(* PLC project Senza_nome, Sconosciuto Senza_nome 1 *)
(* stored: creationDateTime 2020-08-24T19:28:07, modificationDateTime 2020-09-29T15:52:42 *)

FUNCTION_BLOCK TP_WITH_RESET
  VAR_INPUT
    IN : BOOL;
    PT : TIME;
    RESET : BOOL;
  END_VAR
  VAR_OUTPUT
    Q : BOOL;
    ET : TIME := T#0s;
  END_VAR
  VAR
    STATE : SINT := 0;
    PREV_IN : BOOL := FALSE;
    CURRENT_TIME : TIME;
    START_TIME : TIME;
  END_VAR

            (* Pragma to set current time *)
{__SET_VAR(data__->,CURRENT_TIME,,__CURRENT_TIME)}

(*Timer block code *)
IF ((STATE = 0) AND NOT(PREV_IN) AND IN) THEN  (* found rising edge on IN *)
    (* start timer... *)
    STATE := 1;
    Q := TRUE;
    START_TIME := CURRENT_TIME;

ELSIF (STATE = 1) THEN (* timer counting *)
    IF ((START_TIME + PT) <= CURRENT_TIME) THEN (* timer expired *)
        STATE := 2;
        Q := FALSE;
        ET := PT;
    ELSE (* continue counting *)
        ET := CURRENT_TIME - START_TIME;
    END_IF;
END_IF;

IF ((STATE = 2) AND NOT(IN)) THEN
    ET := T#0s;
    STATE := 0;
END_IF;

IF (RESET) THEN (* reset pressed *)
  ET := T#0s;
  STATE := 0;
  Q := FALSE;
END_IF;

PREV_IN := IN;
          
END_FUNCTION_BLOCK

FUNCTION_BLOCK AccensioneProgrammata
  VAR
    TP_WITH_RESET0 : TP_WITH_RESET;  (* Istanza blocco funzionale timer con reset *)
    Aux : BOOL;  (* Variabile ausiliare *)
    Tempo0 : TIME := T#3s;  (* Variabile connessa all'accensione programmata *)
  END_VAR
  VAR_INPUT
    OreDallAccensione : TIME;  (* Associata al PT del secondo timer *)
    Ingresso : BOOL;  (* Variabile di ingresso *)
    Reset : BOOL;  (* Variabile connessa al reset dei timer *)
  END_VAR
  VAR_OUTPUT
    UscitaOn : BOOL;  (* Variabile di uscita *)
  END_VAR
  VAR
    TP_WITH_RESET1 : TP_WITH_RESET;  (* Istanza blocco funzionale timer con reset *)
  END_VAR
  VAR  (* added by the conversion: wires and edge detectors of the diagram *)
    R_TRIG1 : R_TRIG;
    R_TRIG2 : R_TRIG;
    F_TRIG3 : F_TRIG;
  END_VAR

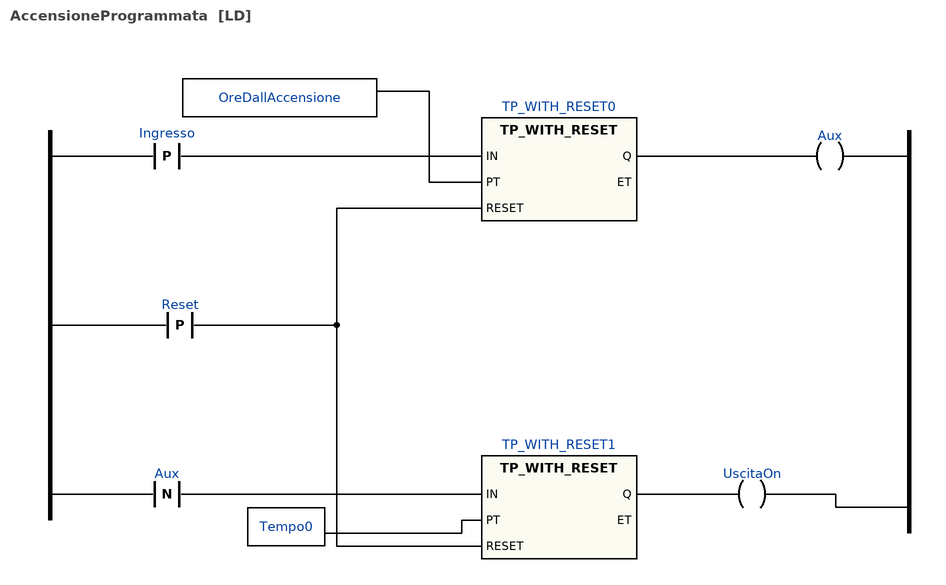
(* LD diagram, written out as Structured Text *)
R_TRIG1(CLK := Ingresso);
R_TRIG2(CLK := Reset);
TP_WITH_RESET0(IN := R_TRIG1.Q, PT := OreDallAccensione, RESET := R_TRIG2.Q);
Aux := TP_WITH_RESET0.Q;
F_TRIG3(CLK := Aux);
TP_WITH_RESET1(IN := F_TRIG3.Q, PT := Tempo0, RESET := R_TRIG2.Q);
UscitaOn := TP_WITH_RESET1.Q;
END_FUNCTION_BLOCK

FUNCTION_BLOCK Macchine
  VAR_INPUT
    TempoDiLavorazione : TIME;  (* Variabile connessa al tempo di lavorazione della macchina *)
    Ingresso : BOOL := 0;  (* Variabile di ingresso *)
    Reset : BOOL := 0;  (* Variabile connessa al reset dei timer *)
  END_VAR
  VAR_OUTPUT
    UscitaMacchina : BOOL := 0;  (* Variabile di uscita *)
  END_VAR
  VAR
    TP_WITH_RESET0 : TP_WITH_RESET;  (* Istanza blocco funzionale timer con reset *)
  END_VAR
  VAR  (* added by the conversion: wires and edge detectors of the diagram *)
    R_TRIG1 : R_TRIG;
    R_TRIG2 : R_TRIG;
  END_VAR

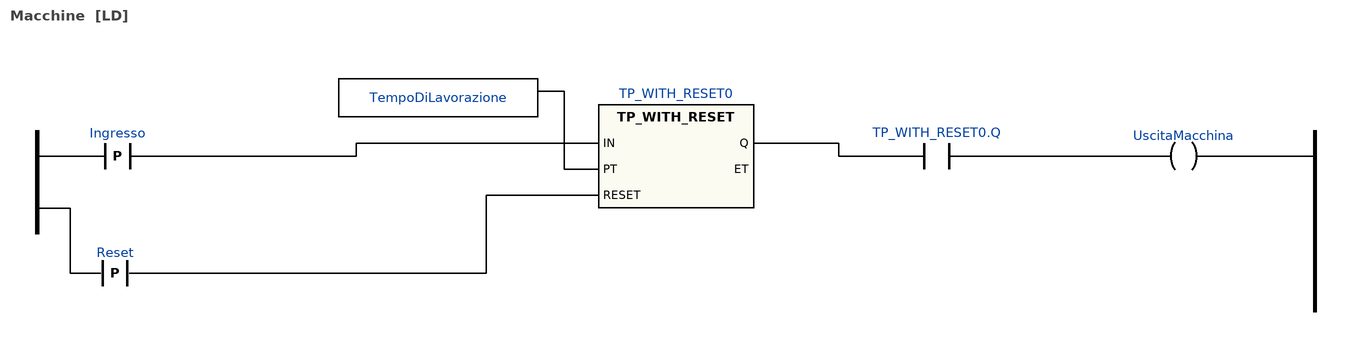
(* LD diagram, written out as Structured Text *)
R_TRIG1(CLK := Ingresso);
R_TRIG2(CLK := Reset);
TP_WITH_RESET0(IN := R_TRIG1.Q, PT := TempoDiLavorazione, RESET := R_TRIG2.Q);
UscitaMacchina := TP_WITH_RESET0.Q AND TP_WITH_RESET0.Q;
END_FUNCTION_BLOCK

FUNCTION_BLOCK Nastro1
  VAR_INPUT
    TempoEsecuzione : TIME;  (* Variabile connessa al tempo di movimento del nastro *)
  END_VAR
  VAR
    TempoInterno : TIME := T#2s;  (* Associata al PT del primo timer *)
  END_VAR
  VAR_INPUT
    Ingresso : BOOL := 0;  (* Variabile di ingresso *)
    reset : BOOL := 0;  (* Variabile connessa al reset dei timer *)
  END_VAR
  VAR_OUTPUT
    UscitaNastro : BOOL := 0;  (* Variabile di uscita *)
  END_VAR
  VAR
    aux : BOOL;  (* Variabile ausiliare *)
    TP_WITH_RESET1 : TP_WITH_RESET;  (* Istanza blocco funzionale timer con reset *)
    TP_WITH_RESET2 : TP_WITH_RESET;  (* Istanza blocco funzionale timer con reset *)
  END_VAR
  VAR  (* added by the conversion: wires and edge detectors of the diagram *)
    R_TRIG1 : R_TRIG;
    R_TRIG2 : R_TRIG;
    F_TRIG3 : F_TRIG;
  END_VAR

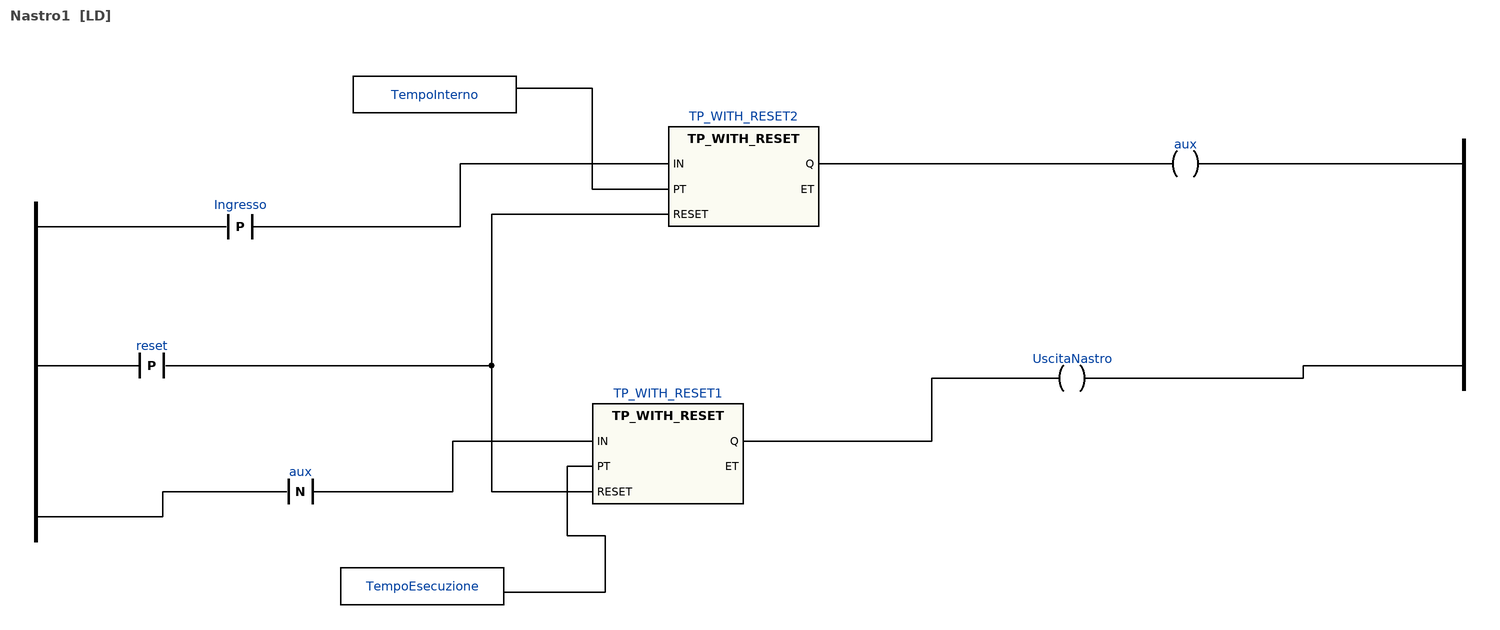
(* LD diagram, written out as Structured Text *)
R_TRIG1(CLK := Ingresso);
R_TRIG2(CLK := reset);
TP_WITH_RESET2(IN := R_TRIG1.Q, PT := TempoInterno, RESET := R_TRIG2.Q);
aux := TP_WITH_RESET2.Q;
F_TRIG3(CLK := aux);
TP_WITH_RESET1(IN := F_TRIG3.Q, PT := TempoEsecuzione, RESET := R_TRIG2.Q);
UscitaNastro := TP_WITH_RESET1.Q;
END_FUNCTION_BLOCK

FUNCTION_BLOCK RisprmioEnergetico
  VAR_OUTPUT
    Uscita : BOOL := 0;  (* Variabile di uscita *)
  END_VAR
  VAR
    aux : BOOL := 0;  (* Variabile ausiliare *)
  END_VAR
  VAR_INPUT
    Ingresso : BOOL := 0;  (* Variabile di ingresso *)
    Reset : BOOL := 0;  (* Variabile connessa al reset dei timer *)
    Tempo : TIME;  (* Associata al PT del primo timer *)
  END_VAR
  VAR
    Tempo2 : TIME := T#4s;  (* Associata al PT del secondo timer *)
    TP_WITH_RESET0 : TP_WITH_RESET;  (* Istanza blocco funzionale timer con reset *)
    TP_WITH_RESET1 : TP_WITH_RESET;  (* Istanza blocco funzionale timer con reset *)
  END_VAR
  VAR  (* added by the conversion: wires and edge detectors of the diagram *)
    R_TRIG1 : R_TRIG;
    F_TRIG2 : F_TRIG;
  END_VAR

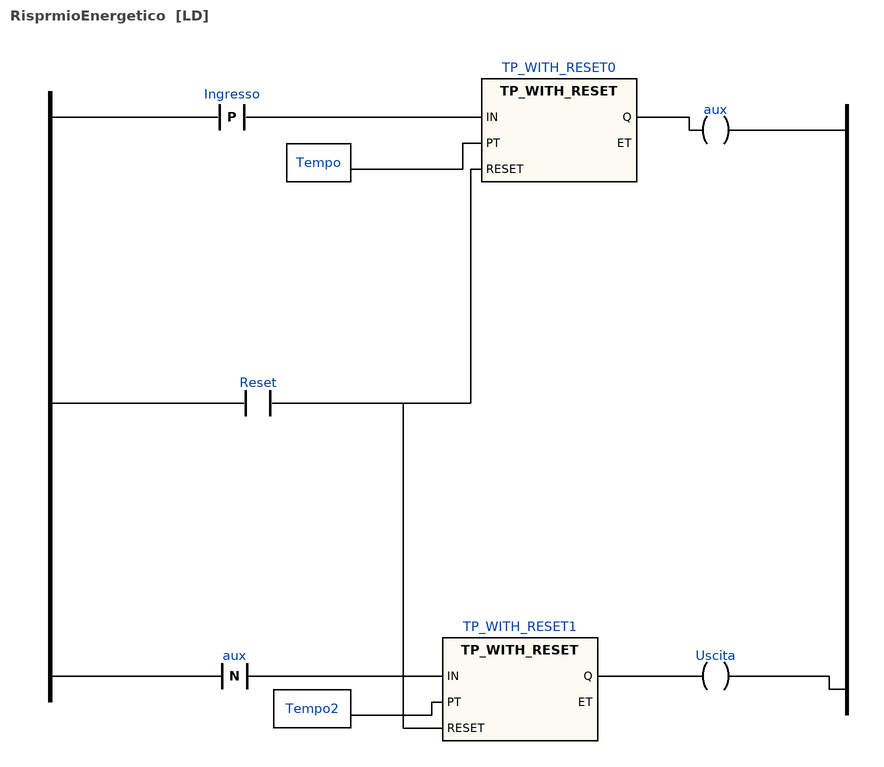
(* LD diagram, written out as Structured Text *)
R_TRIG1(CLK := Ingresso);
TP_WITH_RESET0(IN := R_TRIG1.Q, PT := Tempo, RESET := Reset);
aux := TP_WITH_RESET0.Q;
F_TRIG2(CLK := aux);
TP_WITH_RESET1(IN := F_TRIG2.Q, PT := Tempo2, RESET := Reset);
Uscita := TP_WITH_RESET1.Q;
END_FUNCTION_BLOCK

PROGRAM program0
  VAR
    TastoOn : BOOL := 0;  (* Variabile connessa al pulsante On della macchina *)
  END_VAR
  VAR RETAIN
    AccensioneMan : BOOL := 0;  (* Variabile connessa all'accensione con modalità manuale della macchina *)
    AccensioneAut : BOOL := 0;  (* Variabile connessa all'accensione con modalità automatica della macchina *)
  END_VAR
  VAR
    RipristinoX : BOOL := 0;  (* Replica (per problemi di open plc) il marker di fase della fase Ripristino *)
    RisparmioEnergetico1 : BOOL := 0;  (* Variabile per risparimio energetico 1 *)
    RisparmioEnergetico2 : BOOL := 0;  (* Variabile per risparimio energetico 2 *)
    AttivaReset : BOOL := 0;  (* Attiva il reset del timer *)
    AttivaResetRipr : BOOL := 0;  (* Attiva il reset del timer *)
    AttivaReset0 : BOOL := 0;  (* Attiva il reset del timer *)
    AttivaReset2 : BOOL := 0;  (* Attiva il reset del timer *)
    AttivaReset3 : BOOL := 0;  (* Attiva il reset del timer *)
    AttivaReset4 : BOOL := 0;  (* Attiva il reset del timer *)
    AttivaReset5 : BOOL := 0;  (* Attiva il reset del timer *)
    AttivaReset6 : BOOL := 0;  (* Attiva il reset del timer *)
    AttivaReset7 : BOOL := 0;  (* Attiva il reset del timer *)
    TempoAttesa : BOOL := 0;  (* Sono utilizzate in sostituzione ai timer di fase *)
    TempoAttesa2 : BOOL := 0;  (* Sono utilizzate in sostituzione ai timer di fase *)
    TempoAttesa3 : BOOL := 0;  (* Sono utilizzate in sostituzione ai timer di fase *)
    TimeDummy1 : BOOL := 0;  (* Sono utilizzate in sostituzione ai timer di fase *)
    TimeDummy2 : BOOL := 0;  (* Sono utilizzate in sostituzione ai timer di fase *)
    TimeDummy3 : BOOL := 0;  (* Sono utilizzate in sostituzione ai timer di fase *)
    TimeDummy4 : BOOL := 0;  (* Sono utilizzate in sostituzione ai timer di fase *)
    TimeDummy5 : BOOL := 0;  (* Sono utilizzate in sostituzione ai timer di fase *)
    TimeDummy6 : BOOL := 0;  (* Sono utilizzate in sostituzione ai timer di fase *)
    TimeDummy7 : BOOL := 0;  (* Sono utilizzate in sostituzione ai timer di fase *)
    MacchinaRiscaldata : BOOL := 0;  (* Variabile associata al riscaldamento iniziale della macchina *)
    Time3 : TIME := T#5s;  (* Varibile di tempo utilizzata in Nastro1 e preFineNastro *)
    Time5 : TIME := T#7s;  (* Varibile di tempo utilizzata in fust,Nastro2,StampaAcaldo *)
    Time6 : TIME := T#12s;  (* Varibile di tempo utilizzata in SvuotaNastro *)
    Time7 : TIME := T#900s;  (* Varibile di tempo utilizzata in SvuotaNastro *)
    Time8 : TIME := T#1h;  (* Varibile di tempo utilizzata in SvuotaNastro *)
    Time9 : TIME := T#60s;  (* Varibile di tempo utilizzata in SvuotaNastro *)
  END_VAR
  VAR RETAIN
    TempoProgrammato : TIME := T#0s;  (* Tempo inserito per la futura accensione programmata *)
  END_VAR
  VAR
    LedVerde : BOOL := 0;  (* Variabile connessa al led verde *)
    LedGiallo : BOOL := 0;  (* Variabile connessa al led giallo *)
    LedBianco : BOOL := 0;  (* Variabile connessa al led bianco *)
    ErroreMacchina2 : BOOL := 0;  (* Variabile connessa ad un errore alla macchina che stampa a caldo *)
    ErroreMacchina1 : BOOL := 0;  (* Variabile connessa ad un errore alla macchina che fustella *)
    LedNero : BOOL := 0;  (* Variabile connessa al led nero *)
    LedRosso : BOOL := 0;  (* Variabile connessa al led rosso *)
    TastoCaricoBusta : BOOL := 0;  (* Variabile connessa al pulsante Carico Busta *)
    TastoOff : BOOL := 0;  (* Variabile connessa al pulsante Off della macchina *)
    StartLavorazione : BOOL := 0;  (* Variabile connessa al pulsante Start Lavorazione *)
    Vano : BOOL := 1;  (* Variabile legata al vano di sicurezza della macchina ( gestita in logica negata) *)
    TastoEmergenza : BOOL := 1;  (* Variabile connessa al pulsante di Emergenza della macchina ( gestita in logica negata) *)
    StatoFustellatrice : BOOL := 0;  (* Variabile connessa allo stato della Fustellatrice *)
    StatoStampaACaldo : BOOL := 0;  (* Variabile connessa allo stato della stampa a caldo *)
    Nastro : BOOL := 0;  (* Variabile connessa al nastro trasportatore *)
    SensoreFoil : BOOL := 0;  (* Variabile connessa al sensore del foil (inchiostro) della stampa a caldo *)
    SensoreTemp : BOOL := 0;  (* Variabile connessa al sensore della temperatura della stampa a caldo *)
    SensoreLama : BOOL := 0;  (* Variabile connessa al sensore della lama (indica l'usura) della fustellatrice *)
    RisprmioEnergetico1 : RisprmioEnergetico;  (* Istanza blocco funzionale *)
    RisprmioEnergetico0 : RisprmioEnergetico;  (* Istanza blocco funzionale *)
    Nastro11 : Nastro1;  (* Istanza blocco funzionale *)
    Macchine0 : Macchine;  (* Istanza blocco funzionale *)
    Macchine1 : Macchine;  (* Istanza blocco funzionale *)
    Nastro12 : Nastro1;  (* Istanza blocco funzionale *)
    Nastro10 : Nastro1;  (* Istanza blocco funzionale *)
    AccensioneProgrammata0 : AccensioneProgrammata;  (* Istanza blocco funzionale *)
    Nastro13 : Nastro1;  (* Istanza blocco funzionale *)
    TP0 : TP;
    TP1 : TP;
    RisprmioEnergetico2 : RisprmioEnergetico;
    TP2 : TP;
  END_VAR
  VAR  (* added by the conversion: wires and edge detectors of the diagram *)
    F_TRIG1 : F_TRIG;
    F_TRIG2 : F_TRIG;
  END_VAR

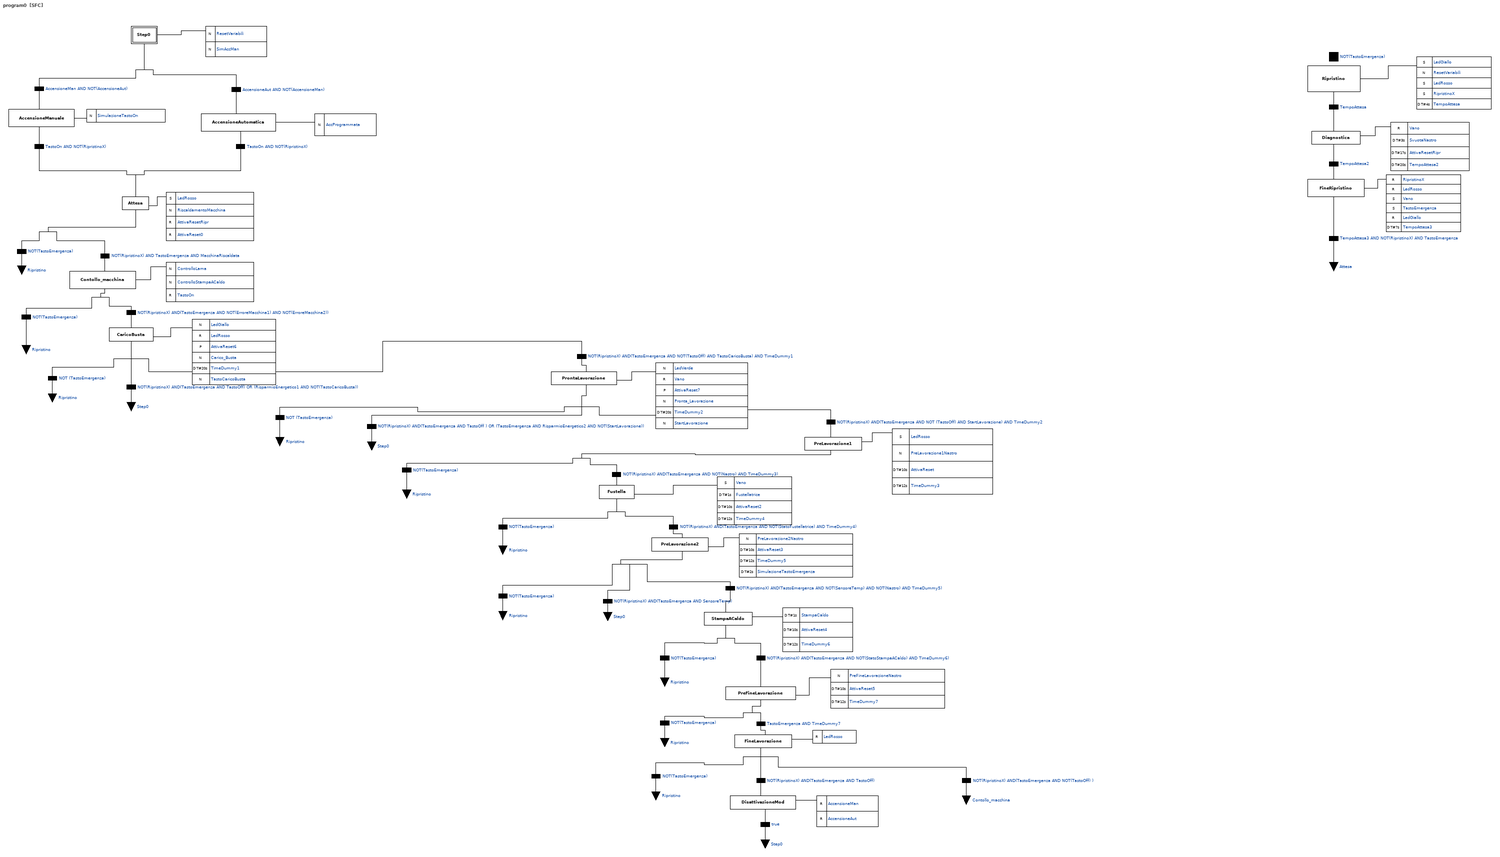
INITIAL_STEP Step0:
  ResetVariabili(N);
  SimAccMan(N);
END_STEP
TRANSITION FROM Step0 TO AccensioneManuale
  := AccensioneMan AND NOT(AccensioneAut);
END_TRANSITION
TRANSITION FROM Step0 TO AccensioneAutomatica
  := AccensioneAut AND NOT(AccensioneMan);
END_TRANSITION
STEP Ripristino:
  LedGiallo(S);
  ResetVariabili(N);
  LedRosso(S);
  RipristinoX(S);
  TempoAttesa(D, T#4s);
END_STEP
TRANSITION FROM Ripristino TO Diagnostica
  := TempoAttesa;
END_TRANSITION
STEP AccensioneManuale:
  SimulazioneTastoOn(N);
END_STEP
TRANSITION FROM AccensioneManuale TO Attesa
  := TastoOn AND NOT(RipristinoX);
END_TRANSITION
STEP AccensioneAutomatica:
  AccProgrammata(N);
END_STEP
TRANSITION FROM AccensioneAutomatica TO Attesa
  := TastoOn AND NOT(RipristinoX);
END_TRANSITION
STEP Diagnostica:
  Vano(R);
  SvuotaNastro(D, T#3s);
  AttivaResetRipr(D, T#17s);
  TempoAttesa2(D, T#20s);
END_STEP
TRANSITION FROM Diagnostica TO FineRipristino
  := TempoAttesa2;
END_TRANSITION
STEP FineRipristino:
  RipristinoX(R);
  LedRosso(R);
  Vano(S);
  TastoEmergenza(S);
  LedGiallo(R);
  TempoAttesa3(D, T#7s);
END_STEP
TRANSITION FROM FineRipristino TO Attesa
  := TempoAttesa3 AND NOT(RipristinoX) AND TastoEmergenza;
END_TRANSITION
STEP Attesa:
  LedRosso(S);
  RiscaldamentoMacchina(N);
  AttivaResetRipr(R);
  AttivaReset0(R);
END_STEP
TRANSITION FROM Attesa TO Ripristino
  := NOT(TastoEmergenza);
END_TRANSITION
TRANSITION FROM Attesa TO Contollo_macchina
  := NOT(RipristinoX) AND TastoEmergenza AND MacchinaRiscaldata;
END_TRANSITION
STEP Contollo_macchina:
  ControlloLama(N);
  ControlloStampaACaldo(N);
  TastoOn(R);
END_STEP
TRANSITION FROM Contollo_macchina TO Ripristino
  := NOT(TastoEmergenza);
END_TRANSITION
TRANSITION FROM Contollo_macchina TO CaricoBusta
  := NOT(RipristinoX) AND(TastoEmergenza AND NOT(ErroreMacchina1) AND NOT(ErroreMacchina2));
END_TRANSITION
STEP CaricoBusta:
  LedGiallo(N);
  LedRosso(R);
  AttivaReset6(P);
  Carico_Busta(N);
  TimeDummy1(D, T#20s);
  TastoCaricoBusta(N);
END_STEP
TRANSITION FROM CaricoBusta TO Ripristino
  := NOT (TastoEmergenza);
END_TRANSITION
TRANSITION FROM CaricoBusta TO Step0
  := NOT(RipristinoX) AND(TastoEmergenza AND TastoOff) OR (RisparmioEnergetico1 AND NOT(TastoCaricoBusta));
END_TRANSITION
TRANSITION FROM CaricoBusta TO ProntaLavorazione
  := NOT(RipristinoX) AND(TastoEmergenza AND NOT(TastoOff) AND TastoCaricoBusta) AND TimeDummy1;
END_TRANSITION
STEP ProntaLavorazione:
  LedVerde(N);
  Vano(R);
  AttivaReset7(P);
  Pronta_Lavorazione(N);
  TimeDummy2(D, T#20s);
  StartLavorazione(N);
END_STEP
TRANSITION FROM ProntaLavorazione TO Ripristino
  := NOT (TastoEmergenza);
END_TRANSITION
TRANSITION FROM ProntaLavorazione TO Step0
  := NOT(RipristinoX) AND(TastoEmergenza AND TastoOff ) OR (TastoEmergenza AND RisparmioEnergetico2 AND NOT(StartLavorazione));
END_TRANSITION
TRANSITION FROM ProntaLavorazione TO PreLavorazione1
  := NOT(RipristinoX) AND(TastoEmergenza AND NOT (TastoOff) AND StartLavorazione) AND TimeDummy2;
END_TRANSITION
STEP PreLavorazione1:
  LedRosso(S);
  PreLavorazione1Nastro(N);
  AttivaReset(D, T#10s);
  TimeDummy3(D, T#12s);
END_STEP
TRANSITION FROM PreLavorazione1 TO Ripristino
  := NOT(TastoEmergenza);
END_TRANSITION
TRANSITION FROM PreLavorazione1 TO Fustella
  := NOT(RipristinoX) AND(TastoEmergenza AND NOT(Nastro) AND TimeDummy3);
END_TRANSITION
STEP Fustella:
  Vano(S);
  Fustellatrice(D, T#1s);
  AttivaReset2(D, T#10s);
  TimeDummy4(D, T#12s);
END_STEP
TRANSITION FROM Fustella TO Ripristino
  := NOT(TastoEmergenza);
END_TRANSITION
TRANSITION FROM Fustella TO PreLavorazione2
  := NOT(RipristinoX) AND(TastoEmergenza AND NOT(StatoFustellatrice) AND TimeDummy4);
END_TRANSITION
STEP PreLavorazione2:
  PreLavorazione2Nastro(N);
  AttivaReset3(D, T#10s);
  TimeDummy5(D, T#12s);
  SimulazioneTastoEmergenza(D, T#2s);
END_STEP
TRANSITION FROM PreLavorazione2 TO Ripristino
  := NOT(TastoEmergenza);
END_TRANSITION
TRANSITION FROM PreLavorazione2 TO StampaACaldo
  := NOT(RipristinoX) AND(TastoEmergenza AND NOT(SensoreTemp) AND NOT(Nastro) AND TimeDummy5);
END_TRANSITION
TRANSITION FROM PreLavorazione2 TO Step0
  := NOT(RipristinoX) AND(TastoEmergenza AND SensoreTemp);
END_TRANSITION
STEP StampaACaldo:
  StampaCaldo(D, T#1s);
  AttivaReset4(D, T#10s);
  TimeDummy6(D, T#12s);
END_STEP
TRANSITION FROM StampaACaldo TO Ripristino
  := NOT(TastoEmergenza);
END_TRANSITION
TRANSITION FROM StampaACaldo TO PreFineLavorazione
  := NOT(RipristinoX) AND(TastoEmergenza AND NOT(StatoStampaACaldo) AND TimeDummy6);
END_TRANSITION
STEP PreFineLavorazione:
  PreFineLavorazioneNastro(N);
  AttivaReset5(D, T#10s);
  TimeDummy7(D, T#12s);
END_STEP
TRANSITION FROM PreFineLavorazione TO FineLavorazione
  := TastoEmergenza AND TimeDummy7;
END_TRANSITION
TRANSITION FROM PreFineLavorazione TO Ripristino
  := NOT(TastoEmergenza);
END_TRANSITION
STEP FineLavorazione:
  LedRosso(R);
END_STEP
TRANSITION FROM FineLavorazione TO Ripristino
  := NOT(TastoEmergenza);
END_TRANSITION
TRANSITION FROM FineLavorazione TO DisattivazioneMod
  := NOT(RipristinoX) AND(TastoEmergenza AND TastoOff);
END_TRANSITION
TRANSITION FROM FineLavorazione TO Contollo_macchina
  := NOT(RipristinoX) AND(TastoEmergenza AND NOT(TastoOff) );
END_TRANSITION
STEP DisattivazioneMod:
  AccensioneMan(R);
  AccensioneAut(R);
END_STEP
TRANSITION FROM DisattivazioneMod TO Step0
  := true;
END_TRANSITION
TRANSITION FROM ? TO ?
  := NOT(TastoEmergenza);
END_TRANSITION

ACTION RiscaldamentoMacchina:
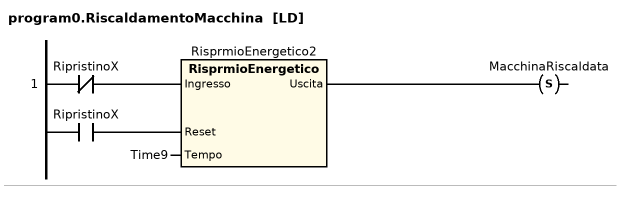
(* LD diagram, written out as Structured Text *)
RisprmioEnergetico2(Ingresso := NOT RipristinoX, Reset := RipristinoX, Tempo := Time9);
IF RisprmioEnergetico2.Uscita THEN MacchinaRiscaldata := TRUE; END_IF;
END_ACTION

ACTION ControlloLama:
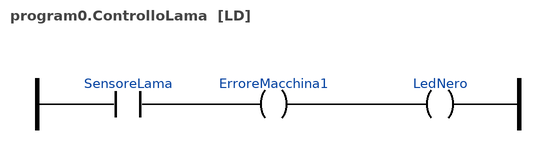
(* LD diagram, written out as Structured Text *)
ErroreMacchina1 := SensoreLama;
LedNero := SensoreLama;
END_ACTION

ACTION ControlloStampaACaldo:
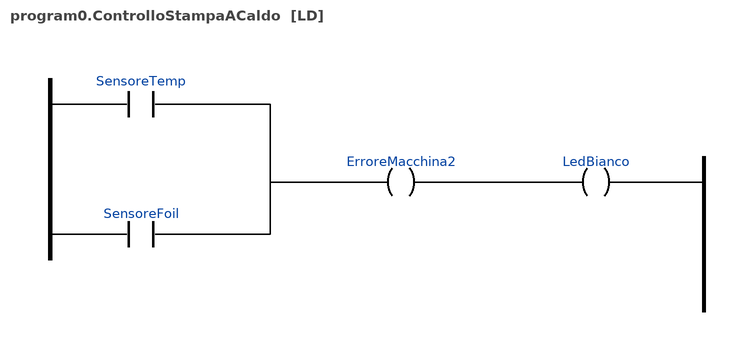
(* LD diagram, written out as Structured Text *)
ErroreMacchina2 := SensoreTemp OR SensoreFoil;
LedBianco := SensoreTemp OR SensoreFoil;
END_ACTION

ACTION Carico_Busta:
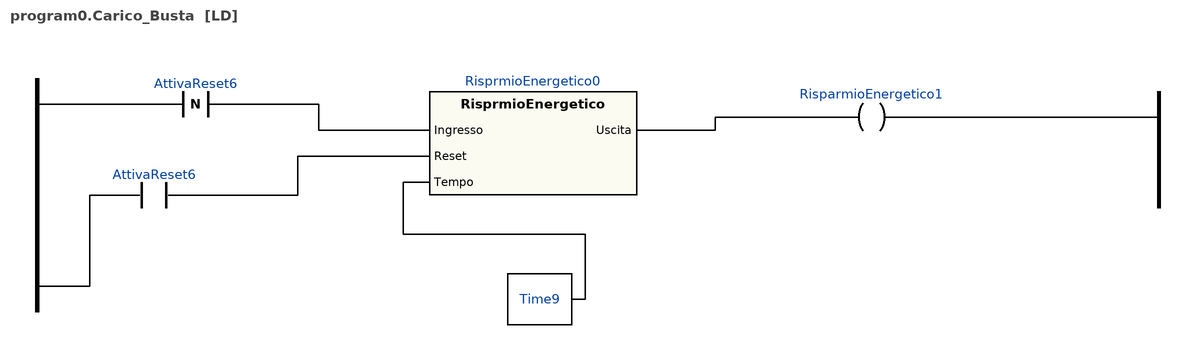
(* LD diagram, written out as Structured Text *)
F_TRIG1(CLK := AttivaReset6);
RisprmioEnergetico0(Ingresso := F_TRIG1.Q, Reset := AttivaReset6, Tempo := Time9);
RisparmioEnergetico1 := RisprmioEnergetico0.Uscita;
END_ACTION

ACTION Pronta_Lavorazione:
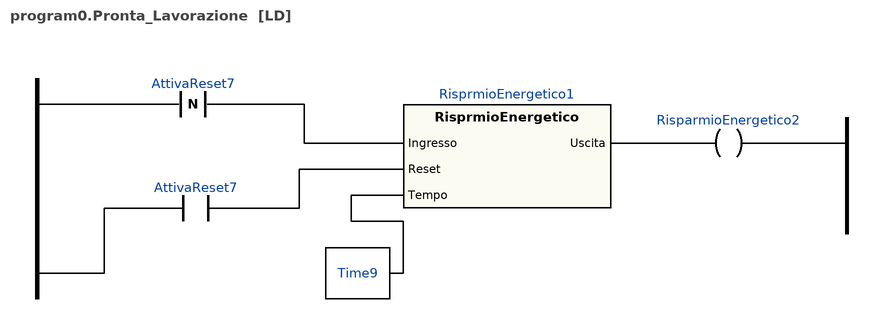
(* LD diagram, written out as Structured Text *)
F_TRIG2(CLK := AttivaReset7);
RisprmioEnergetico1(Ingresso := F_TRIG2.Q, Reset := AttivaReset7, Tempo := Time9);
RisparmioEnergetico2 := RisprmioEnergetico1.Uscita;
END_ACTION

ACTION PreLavorazione1Nastro:
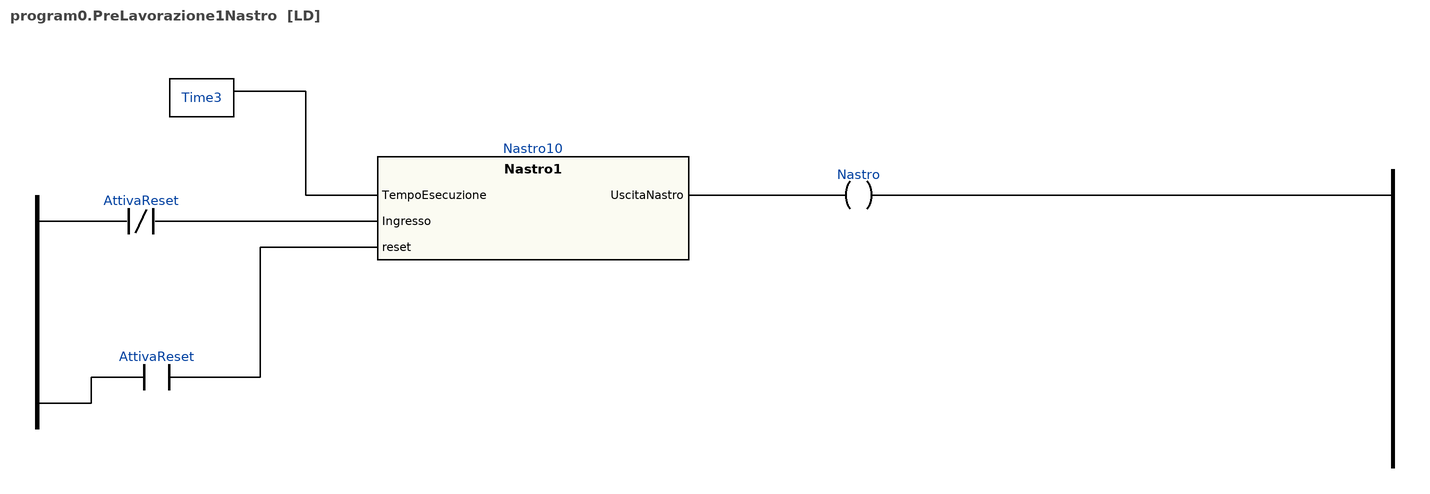
(* LD diagram, written out as Structured Text *)
Nastro10(TempoEsecuzione := Time3, Ingresso := NOT AttivaReset, reset := AttivaReset);
Nastro := Nastro10.UscitaNastro;
END_ACTION

ACTION Fustellatrice:
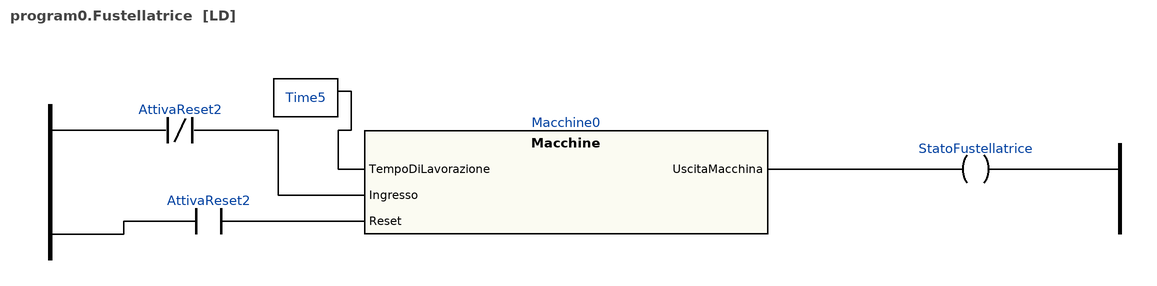
(* LD diagram, written out as Structured Text *)
Macchine0(TempoDiLavorazione := Time5, Ingresso := NOT AttivaReset2, Reset := AttivaReset2);
StatoFustellatrice := Macchine0.UscitaMacchina;
END_ACTION

ACTION PreLavorazione2Nastro:
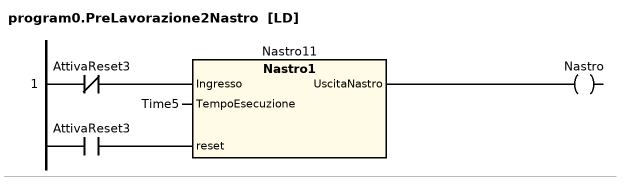
(* LD diagram, written out as Structured Text *)
Nastro11(TempoEsecuzione := Time5, Ingresso := NOT AttivaReset3, reset := AttivaReset3);
Nastro := Nastro11.UscitaNastro;
END_ACTION

ACTION StampaCaldo:
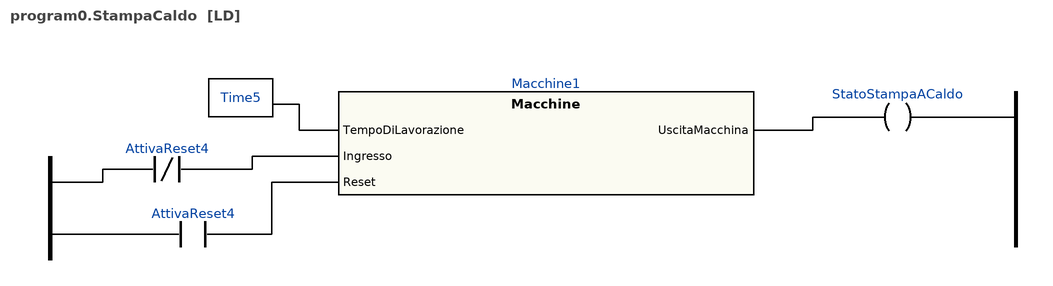
(* LD diagram, written out as Structured Text *)
Macchine1(TempoDiLavorazione := Time5, Ingresso := NOT AttivaReset4, Reset := AttivaReset4);
StatoStampaACaldo := Macchine1.UscitaMacchina;
END_ACTION

ACTION ResetVariabili:
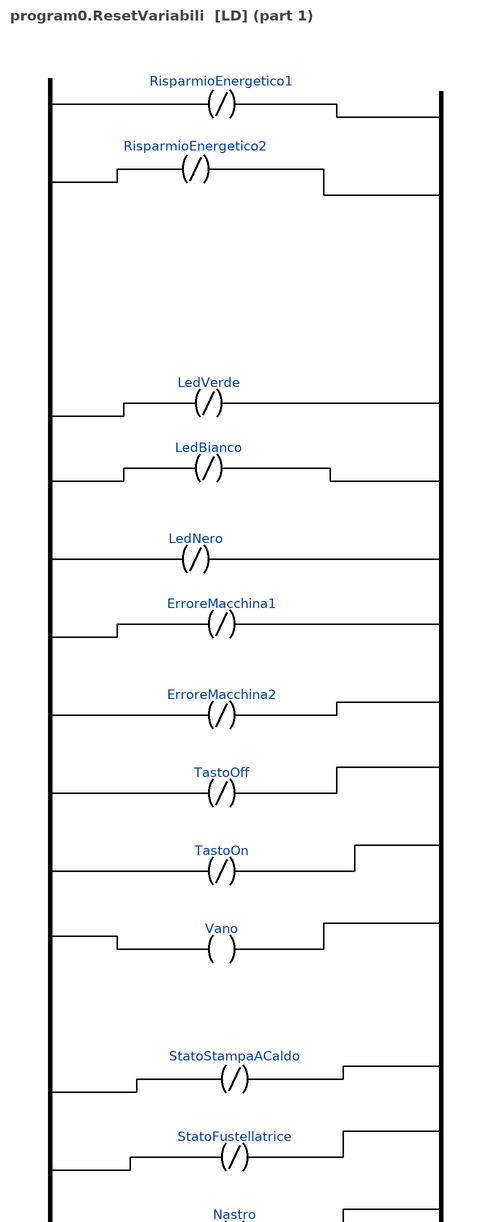
(* LD diagram, written out as Structured Text *)
RisparmioEnergetico1 := NOT TRUE;
RisparmioEnergetico2 := NOT TRUE;
LedVerde := NOT TRUE;
LedBianco := NOT TRUE;
LedNero := NOT TRUE;
ErroreMacchina1 := NOT TRUE;
ErroreMacchina2 := NOT TRUE;
TastoOff := NOT TRUE;
TastoOn := NOT TRUE;
Vano := TRUE;
StatoStampaACaldo := NOT TRUE;
StatoFustellatrice := NOT TRUE;
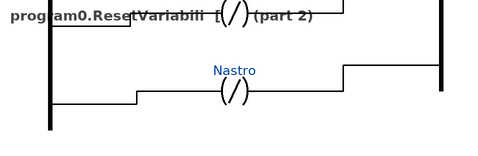
Nastro := NOT TRUE;
END_ACTION

ACTION SpegniRipristino:
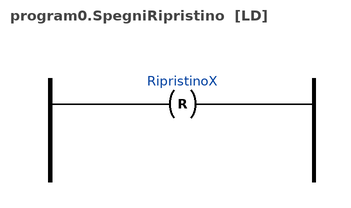
(* LD diagram, written out as Structured Text *)
IF TRUE THEN RipristinoX := FALSE; END_IF;
END_ACTION

ACTION SpegniTasti:
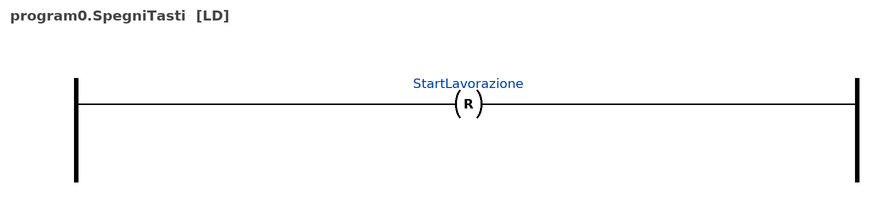
(* LD diagram, written out as Structured Text *)
IF TRUE THEN StartLavorazione := FALSE; END_IF;
END_ACTION

ACTION PreFineLavorazioneNastro:
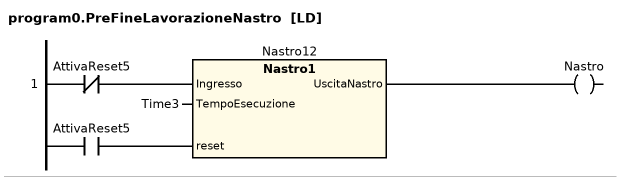
(* LD diagram, written out as Structured Text *)
Nastro12(TempoEsecuzione := Time3, Ingresso := NOT AttivaReset5, reset := AttivaReset5);
Nastro := Nastro12.UscitaNastro;
END_ACTION

ACTION AccProgrammata:
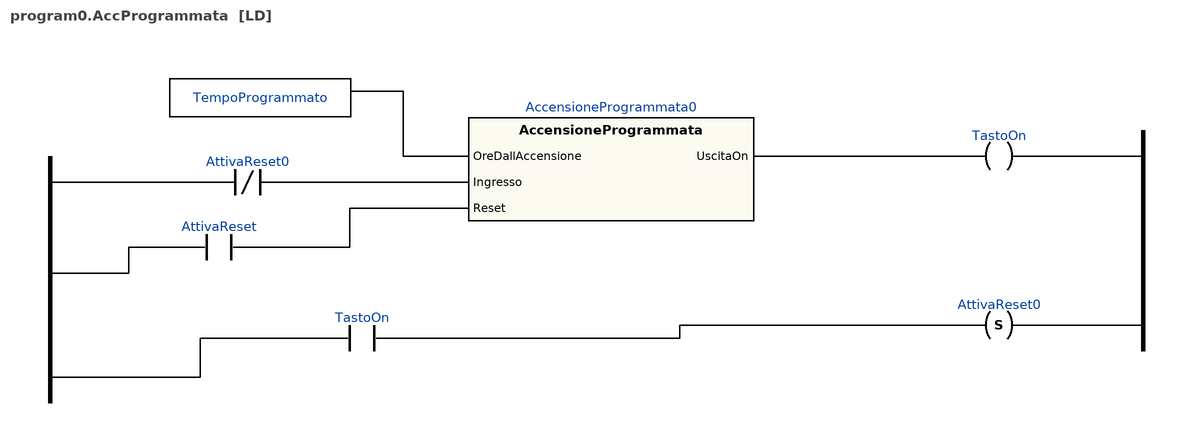
(* LD diagram, written out as Structured Text *)
AccensioneProgrammata0(OreDallAccensione := TempoProgrammato, Ingresso := NOT AttivaReset0, Reset := AttivaReset);
TastoOn := AccensioneProgrammata0.UscitaOn;
IF TastoOn THEN AttivaReset0 := TRUE; END_IF;
END_ACTION

ACTION SimAccMan:
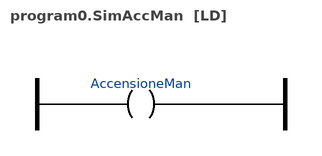
(* LD diagram, written out as Structured Text *)
AccensioneMan := TRUE;
END_ACTION

ACTION SvuotaNastro:
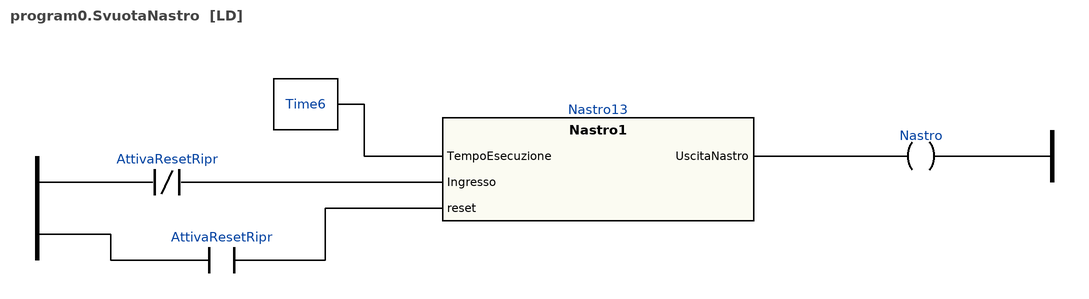
(* LD diagram, written out as Structured Text *)
Nastro13(TempoEsecuzione := Time6, Ingresso := NOT AttivaResetRipr, reset := AttivaResetRipr);
Nastro := Nastro13.UscitaNastro;
END_ACTION

ACTION DisattivazioneModalita:
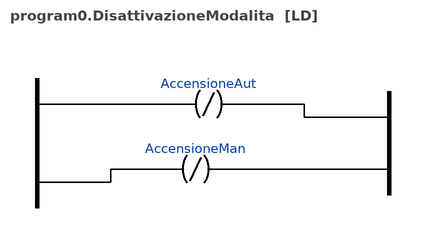
(* LD diagram, written out as Structured Text *)
AccensioneAut := NOT TRUE;
AccensioneMan := NOT TRUE;
END_ACTION

ACTION SimulazioneTastoOn:
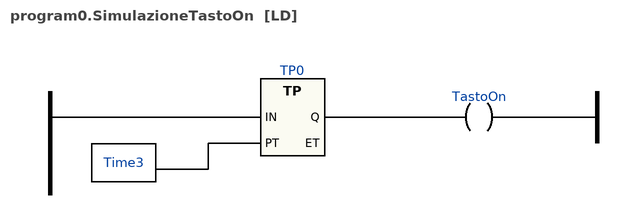
(* LD diagram, written out as Structured Text *)
TP0(IN := TRUE, PT := Time3);
TastoOn := TP0.Q;
END_ACTION

ACTION SimulazioneTastoEmergenza:
